INTERFACE ITF_CUSTOM_TOOL

METHOD Grip : eResult
VAR_INPUT
END_VAR
END_METHOD

PROPERTY Operational : BOOL
SET
END_SET
END_PROPERTY

METHOD Release : eResult
VAR_INPUT
END_VAR
END_METHOD

END_INTERFACE

(* stored: Version 1.1.0.1, ProductVersion 3.1.4026.18
   Itf ITF_CUSTOM_TOOL: Id {e895b00c-8266-4bbf-8de7-8180b6c896da}
   Method Grip: Id {1fe2b9c8-3ecc-4dd9-8c61-eae7e6c9228f}
   Property Operational: Id {fd0de506-4e95-492e-870e-eeeb708f7c63}
   Set Set: Id {5cd67e28-abb9-485b-8a7b-e50851dd6f66}
   Method Release: Id {f0ef0859-c61a-4fd5-9a33-d1f6315a7ca7} *)
